FUNCTION_BLOCK FB_CoE_Read
VAR_INPUT
	// Link this to your terminal's drive reference variables under InfoData.
	stPlcDriveRef : ST_PlcDriveRef;
END_VAR
VAR_OUTPUT
END_VAR
VAR
	// Read Error
	bReadError : BOOL;
	// Data successfully received
	bDataReceived : BOOL := FALSE;
	
	fbCoeRead: FB_CoERead_ByDriveRef;
	
	stDriveRef: ST_DriveRef;
	
	nState : BYTE := 0;   //State Machine
END_VAR

stDriveRef.sNetId := F_CreateAmsNetId(stPlcDriveRef.aNetId);
stDriveRef.nSlaveAddr := stPlcDriveRef.nSlaveAddr;
stDriveRef.nDriveNo := stPlcDriveRef.nDriveNo;
stDriveRef.nDriveType := stPlcDriveRef.nDriveType;

CASE nState OF
	0: //Idle state
		HandleIdle();
	10: //Reading data
		HandleReadingData();
	100: //Handle Error
		HandleError();
END_CASE

ACTION HandleError:
// wait for reset ccmmand
bDataReceived := FALSE;
END_ACTION

ACTION HandleIdle:
fbCoeRead(bExecute := FALSE);
// Reset Data received bit
bDataReceived := FALSE;
END_ACTION

ACTION HandleReadingData:
fbCoeRead(bExecute := TRUE);        // Execute CoE read until done
IF fbCoeRead.bError THEN
	nState := 100;     // Error case
	bReadError := TRUE;
ELSE
	IF NOT fbCoeRead.bBusy THEN
         nState := 0;    // Done
		 bDataReceived := TRUE;
	END_IF
END_IF
END_ACTION

METHOD InErrorState : BOOL
VAR_INPUT
END_VAR
IF nState = 100 THEN
	InErrorState := TRUE;
ELSE
	InErrorState := FALSE;
END_IF
END_METHOD

METHOD IsBusy : BOOL
VAR_INPUT
END_VAR
IF nState <> 0 THEN
	IsBusy := TRUE;
ELSE
	IsBusy := FALSE;
END_IF
END_METHOD

PROPERTY IsDataReceived : BOOL
GET
IsDataReceived := bDataReceived;
END_GET
END_PROPERTY

METHOD ReadData
VAR_INPUT
	//stCoeParameter : ST_CoeParameter;
	nIndex: WORD;
	// Hexadecimal subindex of CoE, e.g. the 12 in 8010:12
	nSubIndex: BYTE;
	// Pointer to a value to fill with the result of the read, e.g. ADR(MyValue)
	pDstBuf: PVOID;
	// Data size of pDstBuf, e.g. SIZEOF(MyValue)
	cbBufLen: UDINT;
END_VAR
IF nState <> 0 THEN
	RETURN;
END_IF

fbCoeRead(
	stDriveRef := stDriveRef,
	nIndex := nIndex,
	nSubIndex := nSubIndex,
	pDstBuf := pDstBuf,
	cbBufLen := cbBufLen,
	tTimeout := T#1S,
);

// Go to Reading data state
nState := 10;
END_METHOD

METHOD ResetError
VAR_INPUT
END_VAR
IF nState <> 100 THEN
	RETURN;
END_IF

// Reset read error
bReadError := FALSE;
// Go to Idle state
nState := 0;
END_METHOD

END_FUNCTION_BLOCK

(* stored: Version 1.1.0.1, ProductVersion 3.1.4022.18
   POU FB_CoE_Read: Id {0468dd5b-db8e-4ac3-9132-a360208fe36e}, SpecialFunc None
   Action HandleError: Id {739f10f7-baba-4f6f-b8d7-517cb0c0f3d5}
   Action HandleIdle: Id {5a4b6f43-8a2e-429c-92c5-ff603e1315c9}
   Action HandleReadingData: Id {9943e26d-2b69-489b-8bb7-40a6a7da0bb3}
   Method InErrorState: Id {872a0ecd-1ce5-4fe0-b2d2-1865bddf380a}
   Method IsBusy: Id {d8e5dfc6-4671-4eb4-af66-9eab1b3b1bb8}
   Property IsDataReceived: Id {b22d3b98-89e5-4f82-a17a-7893834f5f52}
   Get Get: Id {4cc50464-2dbf-4e2e-8aed-cd6e6fdb232a}
   Method ReadData: Id {e9d30cf0-2b10-4894-aa30-a14f26833486}
   Method ResetError: Id {9dcd208a-7420-4c68-8524-06b992b78ef5} *)
